// TIA Portal V16 export
// export: Created 2024-03-28T09:48:20.645095Z, ExportSetting WithDefaults, DisplayName Totally Integrated Automation Portal, DisplayVersion V16, DisplayName TIA Portal Version Control Interface, DisplayVersion V16, DisplayName TIA Portal Openness, DisplayVersion V16, DisplayName STEP 7 Professional, DisplayVersion V16, DisplayName STEP 7 Safety, DisplayVersion V16, DisplayName WinCC Advanced, DisplayVersion V16
TYPE "UR__O2T_IOs"
// stored: IsFailsafeCompliant false
   STRUCT
      "Standard digital output mask" : USInt;
      "Configurable digital output mask" : USInt;
      "Standard digital outputs" : USInt;
      "Configurable digital outputs" : USInt;
      "AOM: Analog output mask" : USInt;
      "AOT: Analog output types" : USInt;
      "TDOM: Tool digital output mask" : USInt;
      "TDO: Tool digital output" : USInt;
      "Standard analog output" : Array[0..1] of Real;
   END_STRUCT;
END_TYPE
